PROGRAM SYSTEM
VAR
END_VAR

GVL.GetLocalSystemTime(
	sNetID := ,
	bEnable := TRUE,
	dwCycle := 1,
	dwOpt:= ,
	tTimeout:= ,
	bValid =>,
	systemTime=>,
	tzID=>);
	
GVL.SystemDateTime := SYSTEMTIME_TO_STRING(GVL.GetLocalSystemTime.systemTime);
GVL.SystemDate := MID(STR:= GVL.SystemDateTime,LEN:=10,POS:=1);
GVL.SystemTime := MID(STR:= GVL.SystemDateTime,LEN:=8,POS:=12);
GVL.SystemSeconds := MID(STR:= GVL.SystemDateTime,LEN:=2,POS:=18);

END_PROGRAM

(* stored: Version 1.1.0.1, ProductVersion 3.1.4024.12
   POU SYSTEM: Id {5993af88-c718-4771-85b6-f8eb292e92b8}, SpecialFunc None *)
